// TwinCAT 3 PLC project Results
// Title: Results
// Company: _
// Author: Krystian Lis et al.
// ProjectVersion: 1.0.0
// Description: Basic result implementation.
// ProgramVersion: 3.1.4026.9
// libraries:
//   Tc3_Module, * (Beckhoff Automation GmbH)
// project tree:
//   Result/Error/ Err.TcGVL, GenericResult.TcGVL
//   Result/ IsErr.TcPOU, IsNone.TcPOU, IsNotNull.TcPOU, IsNull.TcPOU, IsOk.TcPOU, IsSome.TcPOU, Result.TcDUT
// (motion and I/O tree: see PLC project broadcast)
// real-time tasks:
//   TASK PlcTask: cycle T#10ms, priority 20, ADS port 350
//   TASK VISU_TASK: cycle T#200000us, priority 30, ADS port 351

// ---- Result/Result.TcDUT
TYPE Result : INT; END_TYPE

// ---- Result/Error/Err.TcGVL
{attribute 'qualified_only'}
VAR_GLOBAL CONSTANT
	Itf0			: Result := -2;
	Str0			: Result := -3;
	ItfEq			: Result := -4;
	NoMatch			: Result := -5;
	Ptr0			: Result := -6;
	InvRef			: Result := -7;
	Ovf				: Result := -8;
	Udf				: Result := -9;
	Idx				: Result := -10;
	TcLib			: Result := -11;
	InfLoop			: Result := -12;
END_VAR

// ---- Result/Error/GenericResult.TcGVL
VAR_GLOBAL CONSTANT
	None	: Result := 0;
	Ok		: Result := 1;
	Error	: Result := -1;
END_VAR

// ---- Result/IsErr.TcPOU
FUNCTION IsErr : BOOL
VAR_INPUT
	eResult			: Result;
END_VAR
VAR_OUTPUT
	eCarry			: Result;
END_VAR

IsErr := eResult < 0;
eCarry := eResult;

END_FUNCTION

// ---- Result/IsNone.TcPOU
FUNCTION IsNone : BOOL
VAR_INPUT
	eResult			: Result;
END_VAR
VAR_OUTPUT
	eCarry			: Result;
END_VAR

IsNone := eResult = 0;
eCarry := eResult;

END_FUNCTION

// ---- Result/IsNotNull.TcPOU
FUNCTION IsNotNull : BOOL
VAR_INPUT
	anyPtrType		: ANY;
END_VAR

IF anyPtrType.diSize = SIZEOF(POINTER TO BYTE) THEN
	IsNotNull := anyPtrType.pValue^ <> 0;
END_IF

END_FUNCTION

// ---- Result/IsNull.TcPOU
FUNCTION IsNull : BOOL
VAR_INPUT
	anyPtrType		: ANY;
END_VAR

IF anyPtrType.diSize = SIZEOF(POINTER TO BYTE) THEN
	IsNull := anyPtrType.pValue^ = 0;
END_IF

END_FUNCTION

// ---- Result/IsOk.TcPOU
FUNCTION IsOk : BOOL
VAR_INPUT
	eResult			: Result;
END_VAR
VAR_OUTPUT
	eCarry			: Result;
END_VAR

IsOk := eResult > 0;
eCarry := eResult;

END_FUNCTION

// ---- Result/IsSome.TcPOU
FUNCTION IsSome : BOOL
VAR_INPUT
	eResult			: Result;
END_VAR
VAR_OUTPUT
	eCarry			: Result;
END_VAR

IsSome := eResult <> 0;
eCarry := eResult;

END_FUNCTION
